FUNCTION_BLOCK FB_SchedulerAllControl
VAR_INPUT
    bEnableAll : BOOL;   // Toggle all schedulers
END_VAR
VAR_IN_OUT
    FB_Scheduler_F10 : FB_Scheduler_F10;
    FB_Scheduler_F11 : FB_Scheduler_F11; // Extend as needed
    FB_Scheduler_F12 : FB_Scheduler_F12;
END_VAR

END_FUNCTION_BLOCK

(* stored: Version 1.1.0.1, ProductVersion 3.1.4024.14
   POU FB_SchedulerAllControl: Id {6e198c4e-c8c8-4b1e-a3b8-9ce48545d359}, SpecialFunc None *)
